% RSLogix 500 project LEVEL.RSS, saved by version 9.00.00.04 %
PROJECT "PROC1"    % processor: Bul.1763 MicroLogix 1100 Series B %

PROGRAM FILES
  LAD 2 "MAIN"  4 rungs
  LAD 3 "ALARMS"  8 rungs
  LAD 4 "IO"  4 rungs
  LAD 5 "CONTROLS"  6 rungs

DATA FILES
  O0 OUTPUT  5 elements
  I1 INPUT  14 elements
  S2 STATUS  66 elements
  B3 BINARY  1 elements
  T4 TIMER  4 elements
  C5 COUNTER  1 elements
  R6 CONTROL  1 elements
  N7 INTEGER  3 elements
  F8 FLOAT  1 elements

LADDER 2 "MAIN"
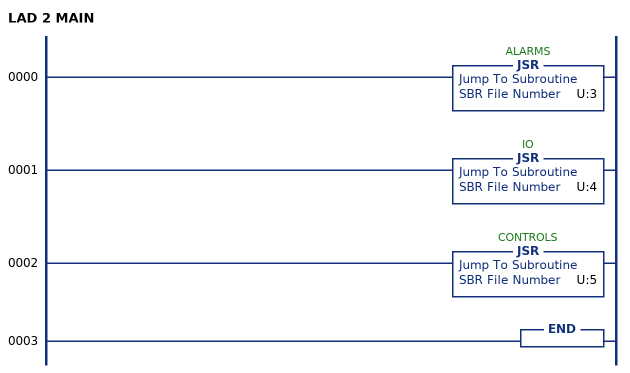
% Rung: 0 %
SOR JSR U:3 EOR
%   U:3  "ALARMS" %
% Rung: 1 %
SOR JSR U:4 EOR
%   U:4  "IO" %
% Rung: 2 %
SOR JSR U:5 EOR
%   U:5  "CONTROLS" %
% Rung: 3 %
SOR END EOR

LADDER 3 "ALARMS"
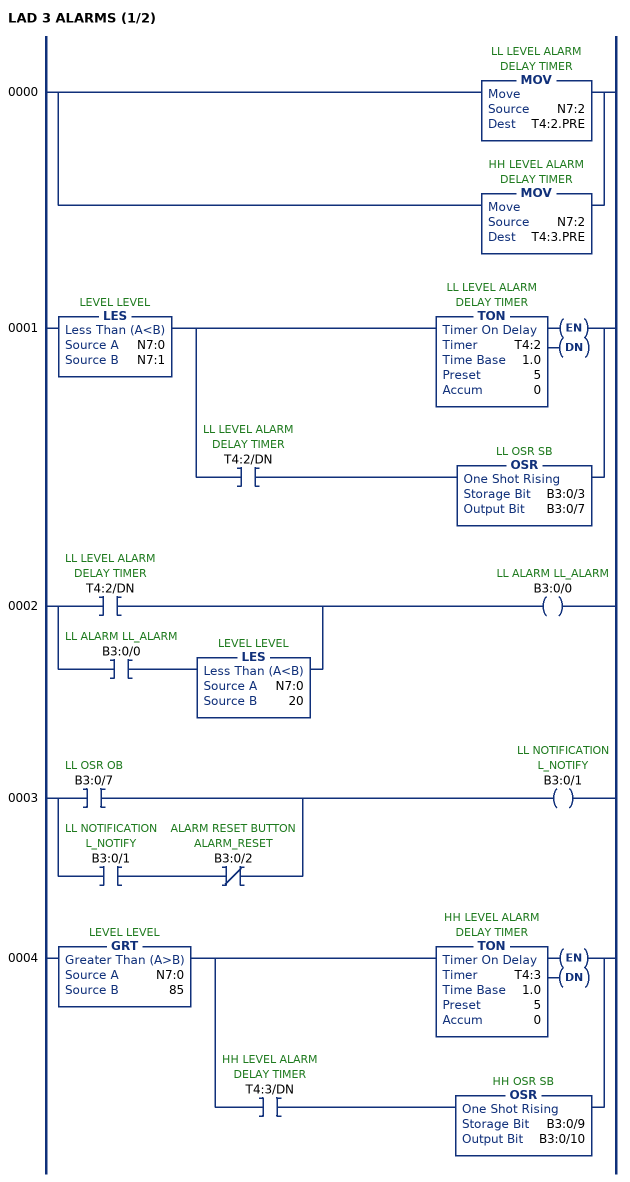
% Rung: 0 %
SOR BST MOV N7:2 T4:2.PRE NXB MOV N7:2 T4:3.PRE BND EOR
%   N7:2  "GENERIC TIME DELAY" %
%   T4:2  "LL LEVEL ALARM DELAY TIMER" %
%   T4:3  "HH LEVEL ALARM DELAY TIMER" %
% Rung: 1 %
SOR LES N7:0 N7:1 BST TON T4:2 1.0 5 0 NXB XIC T4:2/DN OSR B3:0/3 B3:0/7 BND EOR
%   N7:0  LEVEL  "LEVEL" %
%   N7:1  "LL LEVEL SETPOINT FROM HMI" %
%   T4:2  "LL LEVEL ALARM DELAY TIMER" %
%   B3:0/3  "LL OSR SB" %
%   B3:0/7  "LL OSR OB" %
% Rung: 2 %
SOR BST XIC T4:2/DN NXB XIC B3:0/0 LES N7:0 20 BND OTE B3:0/0 EOR
%   T4:2  "LL LEVEL ALARM DELAY TIMER" %
%   B3:0/0  LL_ALARM  "LL ALARM" %
%   N7:0  LEVEL  "LEVEL" %
% Rung: 3 %
SOR BST XIC B3:0/7 NXB XIC B3:0/1 XIO B3:0/2 BND OTE B3:0/1 EOR
%   B3:0/7  "LL OSR OB" %
%   B3:0/1  L_NOTIFY  "LL NOTIFICATION" %
%   B3:0/2  ALARM_RESET  "ALARM RESET BUTTON" %
% Rung: 4 %
SOR GRT N7:0 85 BST TON T4:3 1.0 5 0 NXB XIC T4:3/DN OSR B3:0/9 B3:0/10 BND EOR
%   N7:0  LEVEL  "LEVEL" %
%   T4:3  "HH LEVEL ALARM DELAY TIMER" %
%   B3:0/9  "HH OSR SB" %
%   B3:0/10  "HH OSR OB" %

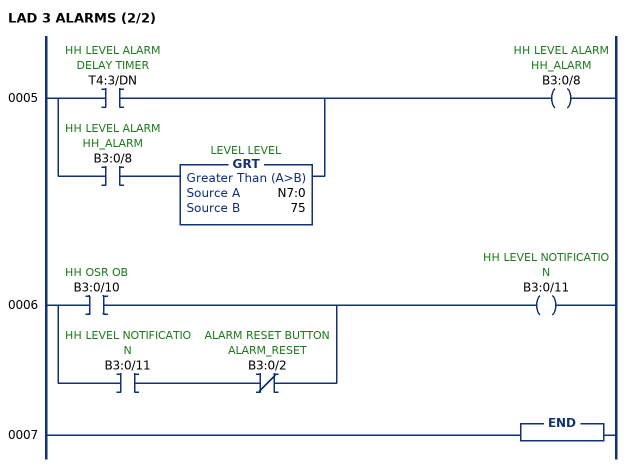
% Rung: 5 %
SOR BST XIC T4:3/DN NXB XIC B3:0/8 GRT N7:0 75 BND OTE B3:0/8 EOR
%   T4:3  "HH LEVEL ALARM DELAY TIMER" %
%   B3:0/8  HH_ALARM  "HH LEVEL ALARM" %
%   N7:0  LEVEL  "LEVEL" %
% Rung: 6 %
SOR BST XIC B3:0/10 NXB XIC B3:0/11 XIO B3:0/2 BND OTE B3:0/11 EOR
%   B3:0/10  "HH OSR OB" %
%   B3:0/11  "HH LEVEL NOTIFICATION" %
%   B3:0/2  ALARM_RESET  "ALARM RESET BUTTON" %
% Rung: 7 %
SOR END EOR

LADDER 4 "IO"
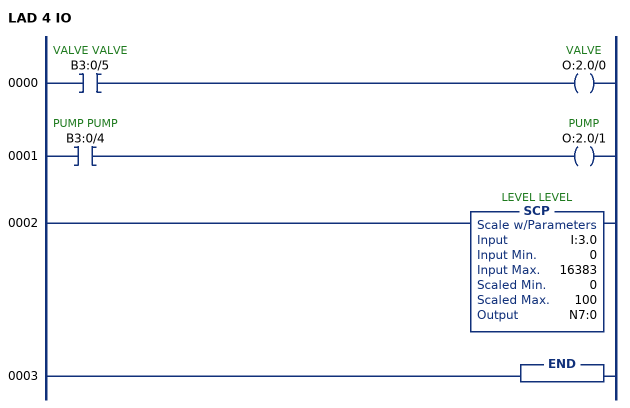
% Rung: 0 %
SOR XIC B3:0/5 OTE O:2.0/0 EOR
%   B3:0/5  VALVE  "VALVE" %
%   O:2.0/0  "VALVE" %
% Rung: 1 %
SOR XIC B3:0/4 OTE O:2.0/1 EOR
%   B3:0/4  PUMP  "PUMP" %
%   O:2.0/1  "PUMP" %
% Rung: 2 %
SOR SCP I:3.0 0 16383 0 100 N7:0 EOR
%   I:3.0  "LEVEL SENSOR INPUT" %
%   N7:0  LEVEL  "LEVEL" %
% Rung: 3 %
SOR END EOR

LADDER 5 "CONTROLS"
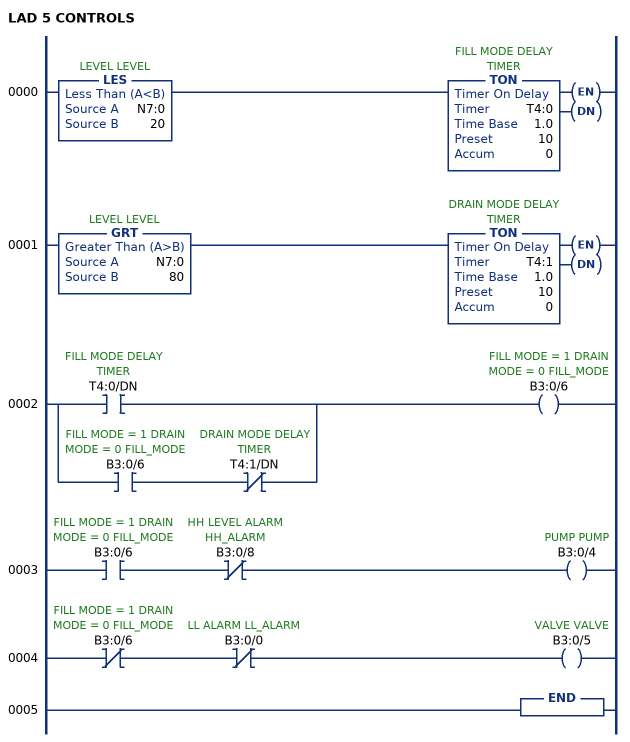
% Rung: 0 %
SOR LES N7:0 20 TON T4:0 1.0 10 0 EOR
%   N7:0  LEVEL  "LEVEL" %
%   T4:0  "FILL MODE DELAY TIMER" %
% Rung: 1 %
SOR GRT N7:0 80 TON T4:1 1.0 10 0 EOR
%   N7:0  LEVEL  "LEVEL" %
%   T4:1  "DRAIN MODE DELAY TIMER" %
% Rung: 2 %
SOR BST XIC T4:0/DN NXB XIC B3:0/6 XIO T4:1/DN BND OTE B3:0/6 EOR
%   T4:0  "FILL MODE DELAY TIMER" %
%   B3:0/6  FILL_MODE  "FILL MODE = 1 DRAIN MODE = 0" %
%   T4:1  "DRAIN MODE DELAY TIMER" %
% Rung: 3 %
SOR XIC B3:0/6 XIO B3:0/8 OTE B3:0/4 EOR
%   B3:0/6  FILL_MODE  "FILL MODE = 1 DRAIN MODE = 0" %
%   B3:0/8  HH_ALARM  "HH LEVEL ALARM" %
%   B3:0/4  PUMP  "PUMP" %
% Rung: 4 %
SOR XIO B3:0/6 XIO B3:0/0 OTE B3:0/5 EOR
%   B3:0/6  FILL_MODE  "FILL MODE = 1 DRAIN MODE = 0" %
%   B3:0/0  LL_ALARM  "LL ALARM" %
%   B3:0/5  VALVE  "VALVE" %
% Rung: 5 %
SOR END EOR

OTHER DOCUMENTED ADDRESSES
  I:1.0/0  "LL SWITCH INPUT"
  I:1.0/1  "L SWITCH INPUT"
  I:1.0/2  "H SWITCH INPUT"
  I:1.0/3  "HH SWITCH INPUT"
  U:6  "ANALOG IO"

REVISION NOTES
  0: TANKPROG

DATA TABLE (non-zero values as saved)
DATA T4
% .PRE .ACC %
% T4:0 % 10 0
% T4:1 % 10 0
% T4:2 % 5 0
% T4:3 % 5 0
